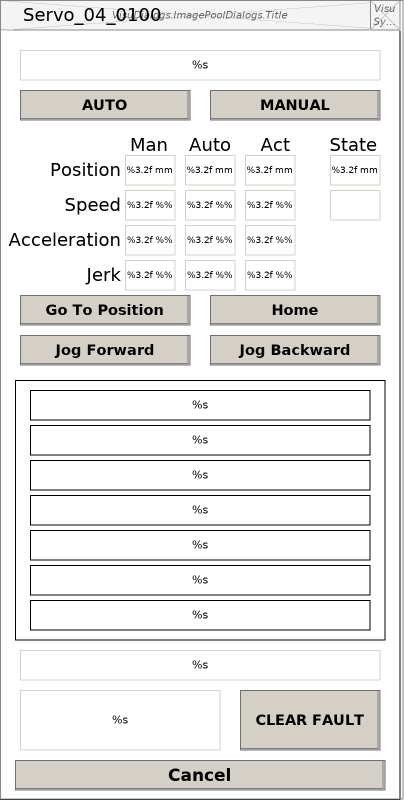
VISUALIZATION visuServoDiag  // 404x800
    Rectangle (0,0 400x800)
    Button (20,90 170x30), "AUTO"
        tap progServoCntrl.Servo_04_0100.AutoReq
    Button (210,90 170x30), "MANUAL"
        tap progServoCntrl.Servo_04_0100.ManReq
    Textfield (20,50 360x30), "%s", text variable: progServoCntrl.Servo_04_0100.strAutoMan
    Image (0,0 400x30), image: VisuDialogs.ImagePoolDialogs.Title
    Group (370,0 30x30)
        RoundedRectangle (0,0 30x30)
        Image (0,0 30x30), image: VisuSymbols.Symbols.Wrong
    Rectangle (15,380 370x260)
    RoundedRectangle (30,390 340x30), "%s", text variable: progSCACntrl.SCA_04_0100.strInterlock_1
    RoundedRectangle (30,425 340x30), "%s", text variable: progSCACntrl.SCA_04_0100.strInterlock_2
    RoundedRectangle (30,460 340x30), "%s", text variable: progSCACntrl.SCA_04_0100.strInterlock_3
    RoundedRectangle (30,495 340x30), "%s", text variable: progSCACntrl.SCA_04_0100.strInterlock_4
    RoundedRectangle (30,530 340x30), "%s", text variable: progSCACntrl.SCA_04_0100.strInterlock_5
    RoundedRectangle (30,565 340x30), "%s", text variable: progSCACntrl.SCA_04_0100.strInterlock_6
    RoundedRectangle (30,600 340x30), "%s", text variable: progSCACntrl.SCA_04_0100.strInterlock_7
    Button (15,760 370x30), "Cancel"
    Label (115,130 56x30), "Man"
    Textfield (125,155 50x30), "%3.2f mm", text variable: progServoCntrl.Servo_04_0100.ManPosSP
        OnMouseClick: write the text variable via VisuDialogs.Numpad, min progSCACntrl.SCA_04_0100.EngMin, max progSCACntrl.SCA_04_0100.EngMax, format %3.2f
    Label (20,0 210x30), "Servo_04_0100"
    Button (20,295 170x30), "Go To Position"
        tap progServoCntrl.Servo_04_0100.GoToPosition
    Textfield (20,650 360x30), "%s", text variable: progServoCntrl.Servo_04_0100.Faulted
    Textfield (20,690 200x60), "%s", text variable: progServoCntrl.Servo_04_0100.FaultID
    Button (240,690 140x60), "CLEAR FAULT"
        tap progServoCntrl.Servo_04_0100.ClearFault
    Label (180,130 54x30), "Auto"
    Label (255,130 38x30), "Act"
    Textfield (125,190 50x30), "%3.2f %%", text variable: progServoCntrl.Servo_04_0100.ManSpeedSP
        OnMouseClick: write the text variable via VisuDialogs.Numpad, min progSCACntrl.SCA_04_0100.EngMin, max progSCACntrl.SCA_04_0100.EngMax, format %3.2f
    Label (45,155 79x30), "Position"
    Label (45,190 79x30), "Speed"
    Label (-4,225 128x30), "Acceleration"
    Label (45,260 79x30), "Jerk"
    Textfield (125,225 50x30), "%3.2f %%", text variable: progServoCntrl.Servo_04_0100.ManAccSP
        OnMouseClick: write the text variable via VisuDialogs.Numpad, min progSCACntrl.SCA_04_0100.EngMin, max progSCACntrl.SCA_04_0100.EngMax, format %3.2f
    Textfield (125,260 50x30), "%3.2f %%", text variable: progServoCntrl.Servo_04_0100.ManJerk
        OnMouseClick: write the text variable via VisuDialogs.Numpad, min progSCACntrl.SCA_04_0100.EngMin, max progSCACntrl.SCA_04_0100.EngMax, format %3.2f
    Textfield (185,155 50x30), "%3.2f mm", text variable: progServoCntrl.Servo_04_0100.AutoPosSp
        OnMouseClick: write the text variable via VisuDialogs.Numpad, min progSCACntrl.SCA_04_0100.EngMin, max progSCACntrl.SCA_04_0100.EngMax, format %3.2f
    Textfield (185,190 50x30), "%3.2f %%", text variable: progServoCntrl.Servo_04_0100.AutoSpeedSp
        OnMouseClick: write the text variable via VisuDialogs.Numpad, min progSCACntrl.SCA_04_0100.EngMin, max progSCACntrl.SCA_04_0100.EngMax, format %3.2f
    Textfield (185,225 50x30), "%3.2f %%", text variable: progServoCntrl.Servo_04_0100.AutoAccSp
        OnMouseClick: write the text variable via VisuDialogs.Numpad, min progSCACntrl.SCA_04_0100.EngMin, max progSCACntrl.SCA_04_0100.EngMax, format %3.2f
    Textfield (185,260 50x30), "%3.2f %%", text variable: progServoCntrl.Servo_04_0100.AutoJerkSp
        OnMouseClick: write the text variable via VisuDialogs.Numpad, min progSCACntrl.SCA_04_0100.EngMin, max progSCACntrl.SCA_04_0100.EngMax, format %3.2f
    Textfield (245,155 50x30), "%3.2f mm", text variable: progServoCntrl.Servo_04_0100.PosSP
        OnMouseClick: write the text variable via VisuDialogs.Numpad, min progSCACntrl.SCA_04_0100.EngMin, max progSCACntrl.SCA_04_0100.EngMax, format %3.2f
    Textfield (245,190 50x30), "%3.2f %%", text variable: progServoCntrl.Servo_04_0100.SpeedSP
        OnMouseClick: write the text variable via VisuDialogs.Numpad, min progSCACntrl.SCA_04_0100.EngMin, max progSCACntrl.SCA_04_0100.EngMax, format %3.2f
    Textfield (245,225 50x30), "%3.2f %%", text variable: progServoCntrl.Servo_04_0100.AccSP
        OnMouseClick: write the text variable via VisuDialogs.Numpad, min progSCACntrl.SCA_04_0100.EngMin, max progSCACntrl.SCA_04_0100.EngMax, format %3.2f
    Textfield (245,260 50x30), "%3.2f %%", text variable: progServoCntrl.Servo_04_0100.JerkSP
        OnMouseClick: write the text variable via VisuDialogs.Numpad, min progSCACntrl.SCA_04_0100.EngMin, max progSCACntrl.SCA_04_0100.EngMax, format %3.2f
    Button (210,295 170x30), "Home"
        tap progServoCntrl.Servo_04_0100.HomeReq
    Button (20,335 170x30), "Jog Forward"
        tap progServoCntrl.Servo_04_0100.JogForward
    Button (210,335 170x30), "Jog Backward"
        tap progServoCntrl.Servo_04_0100.JogBackward
    Label (320,130 60x30), "State"
    Textfield (330,155 50x30), "%3.2f mm", text variable: progServoCntrl.Servo_04_0100.Position
        OnMouseClick: write the text variable via VisuDialogs.Numpad, min progSCACntrl.SCA_04_0100.EngMin, max progSCACntrl.SCA_04_0100.EngMax, format %3.2f
    Textfield (330,190 50x30), text variable: progServoCntrl.Servo_04_0100.Speed
        OnMouseClick: write the text variable via VisuDialogs.Numpad, min progSCACntrl.SCA_04_0100.EngMin, max progSCACntrl.SCA_04_0100.EngMax, format %3.2f
END_VISUALIZATION

(* stored: Version 1.1.0.1, ProductVersion 3.1.4024.6
   Visu visuServoDiag: Id {109fde81-55a5-42fa-b3f5-c0f64a5cb1e4} *)
